Xinje XCPPro project, PLC1: XC3-24 (software 3.3k)

PROGRAM Ladder

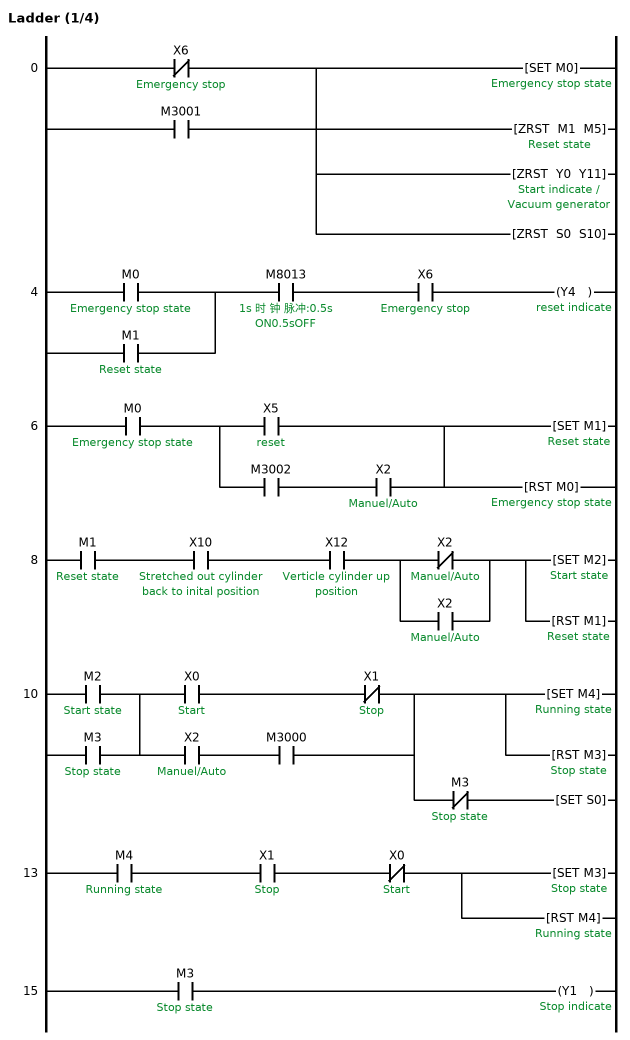
LDI    X6	; Emergency stop
OR     M3001
SET    M0	; Emergency stop state
ZRST   M1 M5	; Reset state
ZRST   Y0 Y11	; Start indicate / Vacuum generator
ZRST   S0 S10
LD     M0	; Emergency stop state
OR     M1	; Reset state
AND    M8013	; 1s 时 钟 脉冲:0.5s ON0.5sOFF
AND    X6	; Emergency stop
OUT    Y4	; reset indicate
LD     M0	; Emergency stop state
LD     X5	; reset
LD     M3002
AND    X2	; Manuel/Auto
ORB
ANB
SET    M1	; Reset state
RST    M0	; Emergency stop state
LD     M1	; Reset state
AND    X10	; Stretched out cylinder back to inital position
AND    X12	; Verticle cylinder up position 
LDI    X2	; Manuel/Auto
OR     X2	; Manuel/Auto
ANB
SET    M2	; Start state
RST    M1	; Reset state
LD     M2	; Start state
OR     M3	; Stop state
LD     X0	; Start
ANI    X1	; Stop
LD     X2	; Manuel/Auto
AND    M3000
ORB
ANB
SET    M4	; Running state
RST    M3	; Stop state
ANI    M3	; Stop state
SET    S0
LD     M4	; Running state
AND    X1	; Stop
ANI    X0	; Start
SET    M3	; Stop state
RST    M4	; Running state
LD     M3	; Stop state
OUT    Y1	; Stop indicate

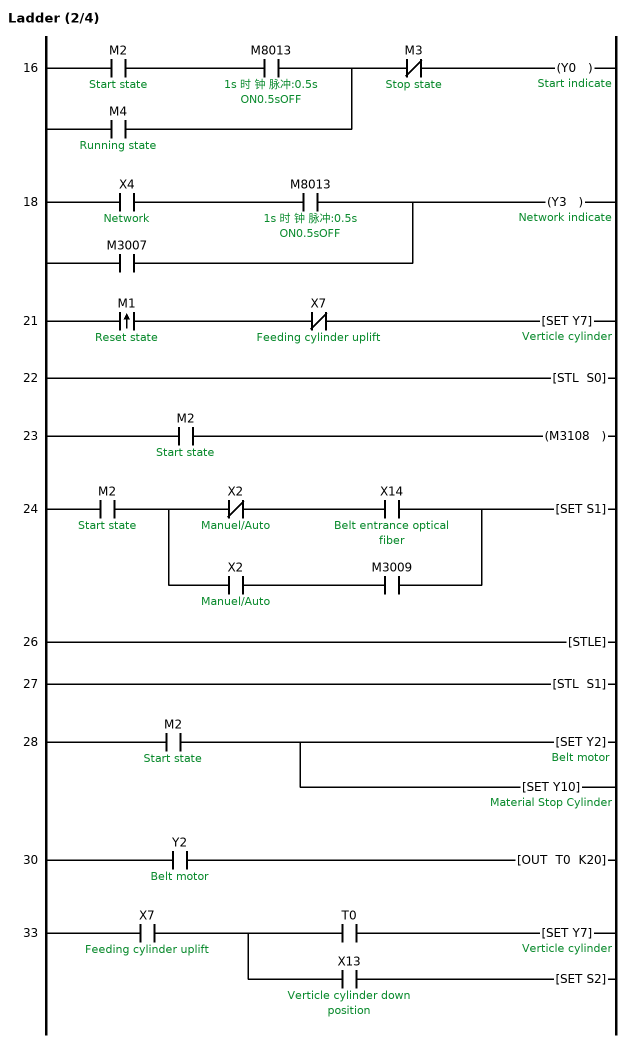
LD     M2	; Start state
AND    M8013	; 1s 时 钟 脉冲:0.5s ON0.5sOFF
OR     M4	; Running state
ANI    M3	; Stop state
OUT    Y0	; Start indicate
LD     X4	; Network
AND    M8013	; 1s 时 钟 脉冲:0.5s ON0.5sOFF
OR     M3007
OUT    Y3	; Network indicate
LDP    M1	; Reset state
ANI    X7	; Feeding cylinder uplift
SET    Y7	; Verticle cylinder
STL    S0
LD     M2	; Start state
OUT    M3108
LD     M2	; Start state
LDI    X2	; Manuel/Auto
AND    X14	; Belt entrance optical fiber
LD     X2	; Manuel/Auto
AND    M3009
ORB
ANB
SET    S1
STLE
STL    S1
LD     M2	; Start state
SET    Y2	; Belt motor
SET    Y10	; Material Stop Cylinder
LD     Y2	; Belt motor
OUT    T0 K20
LD     X7	; Feeding cylinder uplift
MPS
AND    T0
SET    Y7	; Verticle cylinder
MPP
AND    X13	; Verticle cylinder down position 
SET    S2

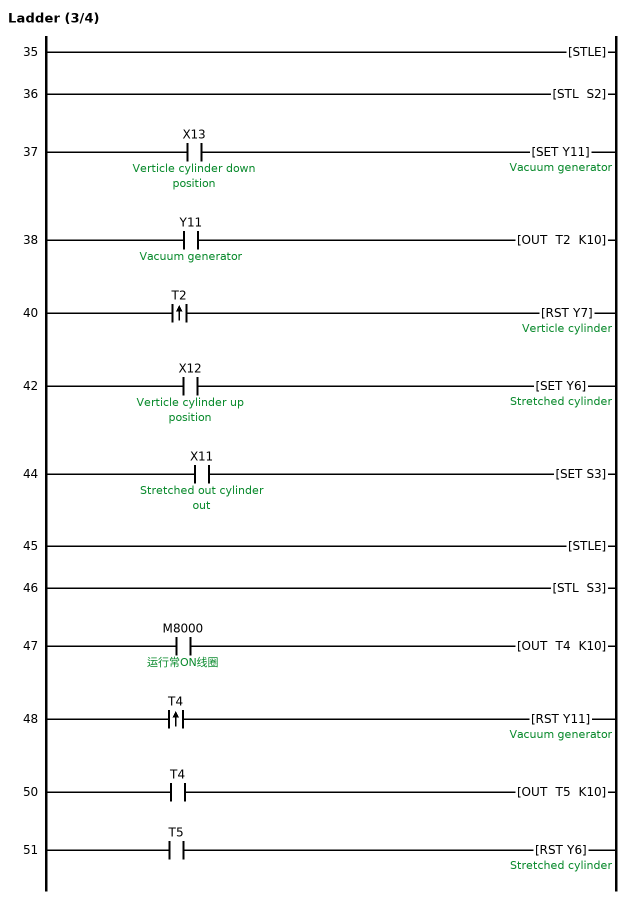
STLE
STL    S2
LD     X13	; Verticle cylinder down position 
SET    Y11	; Vacuum generator
LD     Y11	; Vacuum generator
OUT    T2 K10
LDP    T2
RST    Y7	; Verticle cylinder
LD     X12	; Verticle cylinder up position 
SET    Y6	; Stretched cylinder
LD     X11	; Stretched out cylinder out 
SET    S3
STLE
STL    S3
LD     M8000	; 运行常ON线圈
OUT    T4 K10
LDP    T4
RST    Y11	; Vacuum generator
LD     T4
OUT    T5 K10
LD     T5
RST    Y6	; Stretched cylinder

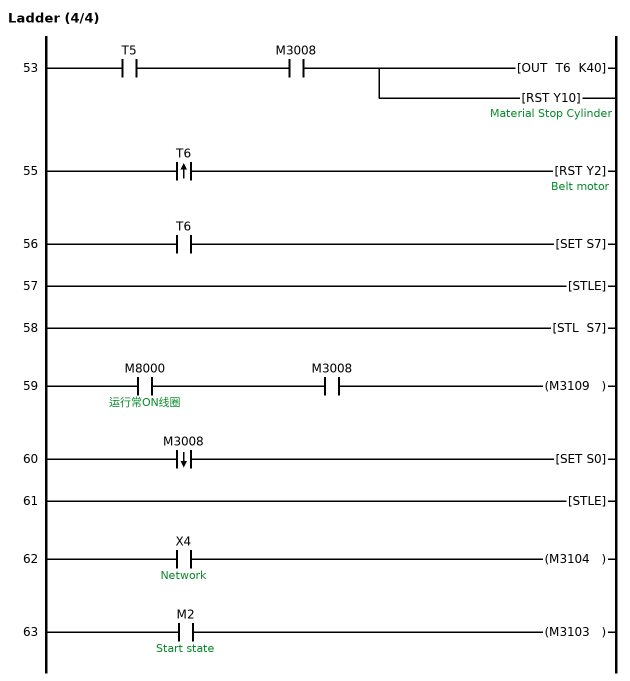
LD     T5
AND    M3008
OUT    T6 K40
RST    Y10	; Material Stop Cylinder
LDP    T6
RST    Y2	; Belt motor
LD     T6
SET    S7
STLE
STL    S7
LD     M8000	; 运行常ON线圈
AND    M3008
OUT    M3109
LDF    M3008
SET    S0
STLE
LD     X4	; Network
OUT    M3104
LD     M2	; Start state
OUT    M3103

COMMENTS (devices not used above)
Y5	Alarm indicate